// SIMATIC S7-200 project (STEP 7-Micro/WIN), CPU 224 REL 02.01

ORGANIZATION_BLOCK MAIN:OB1
TITLE=PROGRAM COMMENTS
BEGIN
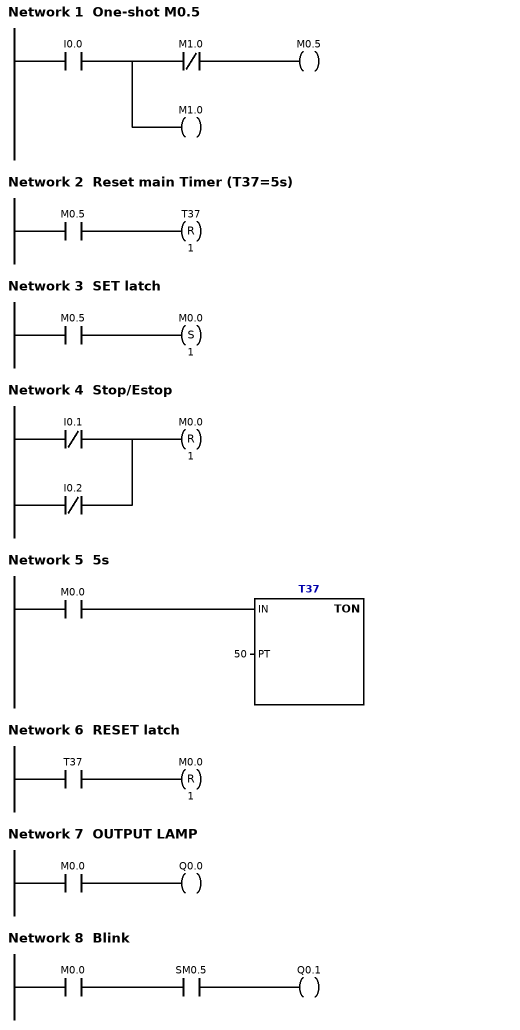
Network 1 // One-shot M0.5
LD     I0.0
LPS
AN     M1.0
=      M0.5
LPP
=      M1.0
Network 2 // Reset main Timer (T37=5s)
LD     M0.5
R      T37, 1
Network 3 // SET latch
LD     M0.5
S      M0.0, 1
Network 4 // Stop/Estop
LDN    I0.1
ON     I0.2
R      M0.0, 1
Network 5 // 5s
LD     M0.0
TON    T37, 50
Network 6 // RESET latch
LD     T37
R      M0.0, 1
Network 7 // OUTPUT LAMP
LD     M0.0
=      Q0.0
Network 8 // Blink
LD     M0.0
A      SM0.5
=      Q0.1
END_ORGANIZATION_BLOCK
